{attribute 'qualified_only'}
VAR_GLOBAL
	Fault: WORD; 
	
	Charging			: BOOL := FALSE;
	Dumping				: BOOL := FALSE;
	ActivateChargePB 	: BOOL := FALSE;
	ActivateDumpPB 		: BOOL := FALSE;
	
END_VAR

(* stored: Version 1.1.0.1, ProductVersion 3.1.4024.9
   GVL HMI_DB: Id {dd8f1866-ff9e-464c-9575-e7dcd895207f} *)
